FUNCTION_BLOCK SAFE_DIV (* Divides two values, clamping on overflow and division-by-zero *)
  (* Standard: 61131-3; Classification: saturating arithmetic function; Description: Copyright (c) 2026 HR Agrartechnik GmbH This program and the accompanying materials are made available under the terms of the Eclipse Public License 2.0 which is available at https://www.eclipse.org/legal/epl-2.0/ SPDX-License-Identifier: EPL-2.0 *)
  (* Version 1.0, 2026-08-27, Franz Höpfinger, HR Agrartechnik GmbH, initial API and implementation and/or initial documentation; division by zero clamps OUT to 0 instead of trapping/producing INF/NaN *)
  PACKAGE SafeArithmetic::arithmetic;
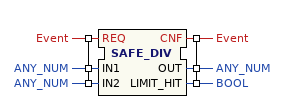
  EVENT_INPUT
    REQ WITH IN1, IN2; (* Normal Execution Request *)
  END_EVENT
  EVENT_OUTPUT
    CNF WITH OUT, LIMIT_HIT; (* Execution Confirmation *)
  END_EVENT
  VAR_INPUT
    IN1 : ANY_NUM; (* First function input (dividend) *)
    IN2 : ANY_NUM; (* Second function input (divisor) *)
  END_VAR
  VAR_OUTPUT
    OUT : ANY_NUM; (* IN1 divided by IN2; 0 if IN2 is 0 *)
    LIMIT_HIT : BOOL; (* TRUE if the result was clamped due to overflow or division by zero *)
  END_VAR
END_FUNCTION_BLOCK
